// TIA Portal V18 export
DATA_BLOCK "DB_Commissioning"   // DB32767
{ S7_Optimized_Access := 'TRUE' }
VERSION : 0.1
// stored: AutoNumber false, DBAccessibleFromOPCUA true, DBAccessibleFromWebserver true, IsOnlyStoredInLoadMemory false, IsRetainMemResEnabled false, IsWriteProtectedInAS false, MemoryReserve 100
   VAR RETAIN
      str : Array[1..8] of String[60];
      bit : Array[1..8] of Bool;
   END_VAR
BEGIN
   str[1] := 'LE4B171420124M33700000131950710';
END_DATA_BLOCK
